PROGRAM tcp_ip
VAR
	bConnect : BOOL;
	bRecieve : BOOL;
	FB_create : FB_SocketUdpCreate;
	FB_Recieve: FB_SocketUdpReceiveFrom;
	FB_close  : FB_SocketClose;
	data: ARRAY[0..5000] OF BYTE;
END_VAR

FB_create(
	sSrvNetId:= , 							//Lokaal netwerk (mag leeg blijven)
	sLocalHost:= '192.168.1.158', 			//Eigen ip van de PC en ingesteld in de gateway
	nLocalPort:= 25565,						//Ingesteld op de gateway
	bExecute:= bConnect,					//Trigger voor functieblok
	tTimeout:= T#10S);


FB_Recieve(
	sSrvNetId:= , 									//Lokaal netwerk (mag leeg blijven)
	hSocket:= FB_create.hSocket,					 
	cbLen:= SIZEOF(data), 							//Kijkt naar de lengte van het bericht
	pDest:= ADR(data), 								//Plaat waar de het bericht wordt opgeslaan
	bExecute:= NOT FB_recieve.bBusy AND bRecieve, 	//Trigger voor functieblok
	tTimeout:= T#10S);
	
FB_close(
	sSrvNetId:= , 							//Lokaal netwerk (mag leeg blijven)
	hSocket:= FB_create.hSocket, 			
	bExecute:= NOT bConnect, 				//Sluiten van de connectie 
	tTimeout:= T#1S);

END_PROGRAM

(* stored: Version 1.1.0.1, ProductVersion 3.1.4024.0
   POU tcp_ip: Id {de64ce75-9f89-4066-b8fa-6c9812ac26d8}, SpecialFunc None *)
